{attribute 'qualified_only'}
{attribute 'strict'}
TYPE eTcoDataFormat : (
    LittleEndian := 1,
    BigEndian := 2
);
END_TYPE

(* stored: Version 1.1.0.1, ProductVersion 3.1.4024.10
   DUT eTcoDataFormat: Id {697416c3-29f9-06b9-3dba-e9f385a30caa} *)
